// TIA Portal V19 export
FUNCTION "FC_Rez_to_DB45" : Void   // FC1, LAD
TITLE = Füllt nach Aufgabetaste (Panel) Technologie DB
{ S7_Optimized_Access := 'TRUE' }
// stored: SetENOAutomatically true
   VAR_TEMP
      Ptr_Befehl_dyn : Int;
      Ptr_Param_dyn : Int;
      i : Int;
   END_VAR
   VAR CONSTANT
      KS : USInt := 1;   // kurz schmal
      LS : USInt := 2;   // lang schmal
      GO : USInt := 3;   // Großoptik
      Typ_KS : Byte := 16#11;
      Typ_LS : Byte := 16#12;
      Typ_GO : Byte := 16#20;
      Startpos_CM01 : Byte := 16#1;
      Startpos_CM02 : Byte := 16#D;
      Startpos_CM03 : Byte := 16#7;
      Startpos_CM04 : Byte := 16#13;
      Startpos_BE : Byte := 16#19;
      Laenge : Byte := 16#6;
      leer : Byte;
      M_area : Byte := 16#83;
      DB_area : Byte := 16#84;
      Ptr_Befehl_1 : Int := 260;   // Adresse Befehlsparameter
      Ptr_Befehl_2 : Int := 264;   // Adresse Befehlsparameter
      Ptr_Befehl_3 : Int := 268;   // Adresse Befehlsparameter
      Ptr_Befehl_4 : Int := 272;   // Adresse Befehlsparameter
      Ptr_Befehl_5 : Int := 276;   // Adresse Befehlsparameter
      Ptr_Befehl_6 : Int := 280;   // Adresse Befehlsparameter
      Ptr_Befehl_7 : Int;   // Adresse Befehlsparameter
      Techno_DB : DInt := 45;
   END_VAR
BEGIN

REGION Network 1 (SCL): aktuelle Auswahl in Arbeitsstruktur kopieren
   IF "DB_Prog_edit".akt_Aufgabe_Prog <> "DB_Prog_edit".old_Aufgabe_Prog THEN
       "DB_Prog_edit".Prog_Aufgabe.Prog := "DB_Prog_edit".Prog["DB_Prog_edit".akt_Aufgabe_Prog];

       "DB_Prog_edit".old_Aufgabe_Prog := "DB_Prog_edit".akt_Aufgabe_Prog;
   END_IF;
END_REGION

REGION Network 2 (SCL): Artikeldaten für aufgabe aufbereiten
   IF "Panel".Aufgabe.Freigabe AND "DB_Prog_edit".StandNr <> 0  AND "DB_Prog_edit".akt_Aufgabe_Prog <>0  AND "DB_Prog_edit".Prog_Aufgabe.Korb_Nr <>0 THEN

       "DB_Prog_edit".GZ_Charge := "DB_Prog_edit".GZ_Charge + 1; // Gesamtzähler erhöhen
       "DB_Techno".WT_NR_lng := "DB_Prog_edit".GZ_Charge; // Chargenzähler
       "DB_Techno".STAND_NR := "DB_Prog_edit".StandNr; // Nummer B/E-Stand: 1..6
       "DB_Techno".Korb_Nr := INT_TO_USINT("DB_Prog_edit".Prog_Aufgabe.Korb_Nr); // Korb 1..13

       // Modus auswerten
       IF NOT "DB_ANLAGE".config.NormalB THEN
           // Kombi-Mode
           CASE "DB_Prog_edit".Prog_Aufgabe.Korb_Nr OF
               1..3:  // "151" Korb kurz 1..3
                   "DB_Prog_edit".Prog_Aufgabe.Prog.ParaByte.%X4 := TRUE;
                   "DB_Prog_edit".Prog_Aufgabe.Prog.ParaByte.%X5 := FALSE;

               4..8:   // "161" Korb kurz 4..8
                   "DB_Prog_edit".Prog_Aufgabe.Prog.ParaByte.%X4 := FALSE;
                   "DB_Prog_edit".Prog_Aufgabe.Prog.ParaByte.%X5 := TRUE;

               9..11:  // "151" Korb lang 1..3
                   "DB_Prog_edit".Prog_Aufgabe.Prog.ParaByte.%X4 := TRUE;
                   "DB_Prog_edit".Prog_Aufgabe.Prog.ParaByte.%X5 := FALSE;

               12..13:   // "161" Korb lang 4, Großoptik 
                   "DB_Prog_edit".Prog_Aufgabe.Prog.ParaByte.%X4 := FALSE;
                   "DB_Prog_edit".Prog_Aufgabe.Prog.ParaByte.%X5 := TRUE;
           END_CASE;

       ELSE
           // Normalbetrieb
           "DB_Prog_edit".Prog_Aufgabe.Prog.ParaByte.%X4 := FALSE;
           "DB_Prog_edit".Prog_Aufgabe.Prog.ParaByte.%X5 := FALSE;
       END_IF;

       "DB_Techno".Technologie := "DB_Prog_edit".akt_Aufgabe_Prog; // aktuelles Programm: 1..99
           // WT-Typ
       CASE "DB_Prog_edit".Prog_Aufgabe.Prog.Geometrie OF
           #KS:  
               "DB_Techno".WT_Typ := #Typ_KS;
           #LS:  
               "DB_Techno".WT_Typ := #Typ_LS;
           #GO:
               "DB_Techno".WT_Typ := #Typ_GO;
           ELSE
               "DB_Techno".WT_Typ := 0;
       END_CASE;
    // Langsam senken /Langsam heben / Modi
       "DB_Techno".ParaByte := "DB_Prog_edit".Prog_Aufgabe.Prog.ParaByte;

       "DB_Techno".KorrATZ := "DB_Prog_edit".Prog_Aufgabe.Prog.Faktor_ATZ;
       "DB_Techno".KorrPend := 1.0;


       // Normal-Betrieb - nur Ware "151" Gruppe CM01/CM02
       IF "DB_ANLAGE".config.NormalB THEN
           REGION NormalB
               // Vorspülen
               #Ptr_Befehl_dyn := 1;
               #Ptr_Param_dyn := 340;

               "DB_Techno".stBefehle[#Ptr_Befehl_dyn].Kennung := #Startpos_CM03;
               "DB_Techno".stBefehle[#Ptr_Befehl_dyn].FirstPos1 := #Startpos_CM03;
               "DB_Techno".stBefehle[#Ptr_Befehl_dyn].Grpleng1 := #Laenge;
               "DB_Techno".stBefehle[#Ptr_Befehl_dyn].FirstPos2 := #leer;
               "DB_Techno".stBefehle[#Ptr_Befehl_dyn].Grpleng2 := #leer;
               "DB_Techno".stBefehle[#Ptr_Befehl_dyn].Merker := #leer;
               "DB_Techno".stBefehle[#Ptr_Befehl_dyn].Param_Ptr := #Ptr_Param_dyn; //#Ptr_Befehl_1;
               "temp_Sollzeit" := TOD_TO_DINT("DB_Prog_edit".Prog_Aufgabe.Prog.CM03_VorSpuel.Expo) / 1000;

               POKE_BLK(area_src := #M_area,
                        dbNumber_src := 0,
                        byteOffset_src := 256,
                        area_dest := #DB_area,
                        dbNumber_dest := #Techno_DB,
                        byteOffset_dest := #Ptr_Param_dyn, //Ptr_Befehl_1,
                        count := 4);

               // Vorätzen
               IF "DB_Prog_edit".Prog_Aufgabe.Prog.CM01_VorAetz.Anzahl_Voraetz > 0 THEN
                   FOR #i := 1 TO BYTE_TO_INT("DB_Prog_edit".Prog_Aufgabe.Prog.CM01_VorAetz.Anzahl_Voraetz) DO
                       #Ptr_Befehl_dyn := #Ptr_Befehl_dyn + 1;
                       #Ptr_Param_dyn := #Ptr_Param_dyn + 4;

                       "DB_Techno".stBefehle[#Ptr_Befehl_dyn].Kennung := #Startpos_CM01;
                       "DB_Techno".stBefehle[#Ptr_Befehl_dyn].FirstPos1 := #Startpos_CM01;
                       "DB_Techno".stBefehle[#Ptr_Befehl_dyn].Grpleng1 := #Laenge;
                       "DB_Techno".stBefehle[#Ptr_Befehl_dyn].FirstPos2 := #Startpos_CM02;
                       "DB_Techno".stBefehle[#Ptr_Befehl_dyn].Grpleng2 := #Laenge;
                       "DB_Techno".stBefehle[#Ptr_Befehl_dyn].Merker := #leer;
                       "DB_Techno".stBefehle[#Ptr_Befehl_dyn].Param_Ptr := #Ptr_Param_dyn; // #Ptr_Befehl_2;
                       "temp_Sollzeit" := TOD_TO_DINT("DB_Prog_edit".Prog_Aufgabe.Prog.CM01_VorAetz.Expo) / 1000;

                       POKE_BLK(area_src := #M_area,
                                dbNumber_src := 0,
                                byteOffset_src := 256,
                                area_dest := #DB_area,
                                dbNumber_dest := #Techno_DB,
                                byteOffset_dest := #Ptr_Param_dyn, //Ptr_Befehl_2,
                                count := 4);


                       // Spülen Vorätzen
                       #Ptr_Befehl_dyn := #Ptr_Befehl_dyn + 1;
                       #Ptr_Param_dyn := #Ptr_Param_dyn + 4;

                       "DB_Techno".stBefehle[#Ptr_Befehl_dyn].Kennung := #Startpos_CM03;
                       "DB_Techno".stBefehle[#Ptr_Befehl_dyn].FirstPos1 := #Startpos_CM03;
                       "DB_Techno".stBefehle[#Ptr_Befehl_dyn].Grpleng1 := #Laenge;
                       "DB_Techno".stBefehle[#Ptr_Befehl_dyn].FirstPos2 := #leer;
                       "DB_Techno".stBefehle[#Ptr_Befehl_dyn].Grpleng2 := #leer;
                       "DB_Techno".stBefehle[#Ptr_Befehl_dyn].Merker := #leer;
                       "DB_Techno".stBefehle[#Ptr_Befehl_dyn].Param_Ptr := #Ptr_Param_dyn; // #Ptr_Befehl_3;
                       "temp_Sollzeit" := TOD_TO_DINT("DB_Prog_edit".Prog_Aufgabe.Prog.CM03_SpuelVorAetz.Expo) / 1000;

                       POKE_BLK(area_src := #M_area,
                                dbNumber_src := 0,
                                byteOffset_src := 256,
                                area_dest := #DB_area,
                                dbNumber_dest := #Techno_DB,
                                byteOffset_dest := #Ptr_Param_dyn, //#Ptr_Befehl_3,
                                count := 4);

                   END_FOR;
               END_IF;

               // Ätzen
               #Ptr_Befehl_dyn := #Ptr_Befehl_dyn + 1;
               #Ptr_Param_dyn := #Ptr_Param_dyn + 4;

               "DB_Techno".stBefehle[#Ptr_Befehl_dyn].Kennung := #Startpos_CM01;
               "DB_Techno".stBefehle[#Ptr_Befehl_dyn].FirstPos1 := #Startpos_CM01;
               "DB_Techno".stBefehle[#Ptr_Befehl_dyn].Grpleng1 := #Laenge;
               "DB_Techno".stBefehle[#Ptr_Befehl_dyn].FirstPos2 := #Startpos_CM02;
               "DB_Techno".stBefehle[#Ptr_Befehl_dyn].Grpleng2 := #Laenge;
               "DB_Techno".stBefehle[#Ptr_Befehl_dyn].Merker := #leer;
               "DB_Techno".stBefehle[#Ptr_Befehl_dyn].Param_Ptr := #Ptr_Param_dyn; //#Ptr_Befehl_4;
               "temp_Sollzeit" := TOD_TO_DINT("DB_Prog_edit".Prog_Aufgabe.Prog.CM01_Aetzen.Expo) / 1000;

               POKE_BLK(area_src := #M_area,
                        dbNumber_src := 0,
                        byteOffset_src := 256,
                        area_dest := #DB_area,
                        dbNumber_dest := #Techno_DB,
                        byteOffset_dest := #Ptr_Param_dyn, //#Ptr_Befehl_4,
                        count := 4);

               // Spülen 1 Ätzen
               #Ptr_Befehl_dyn := #Ptr_Befehl_dyn + 1;
               #Ptr_Param_dyn := #Ptr_Param_dyn + 4;

               "DB_Techno".stBefehle[#Ptr_Befehl_dyn].Kennung := #Startpos_CM03;
               "DB_Techno".stBefehle[#Ptr_Befehl_dyn].FirstPos1 := #Startpos_CM03;
               "DB_Techno".stBefehle[#Ptr_Befehl_dyn].Grpleng1 := #Laenge;
               "DB_Techno".stBefehle[#Ptr_Befehl_dyn].FirstPos2 := #leer;
               "DB_Techno".stBefehle[#Ptr_Befehl_dyn].Grpleng2 := #leer;
               "DB_Techno".stBefehle[#Ptr_Befehl_dyn].Merker := #leer;
               "DB_Techno".stBefehle[#Ptr_Befehl_dyn].Param_Ptr := #Ptr_Param_dyn; //#Ptr_Befehl_5;
               "temp_Sollzeit" := TOD_TO_DINT("DB_Prog_edit".Prog_Aufgabe.Prog.CM03_Spl_1.Expo) / 1000;

               POKE_BLK(area_src := #M_area,
                        dbNumber_src := 0,
                        byteOffset_src := 256,
                        area_dest := #DB_area,
                        dbNumber_dest := #Techno_DB,
                        byteOffset_dest := #Ptr_Param_dyn, //#Ptr_Befehl_5,
                        count := 4);

               // Spülen 2 Ätzen
               #Ptr_Befehl_dyn := #Ptr_Befehl_dyn + 1;
               #Ptr_Param_dyn := #Ptr_Param_dyn + 4;

               "DB_Techno".stBefehle[#Ptr_Befehl_dyn].Kennung := #Startpos_CM04;
               "DB_Techno".stBefehle[#Ptr_Befehl_dyn].FirstPos1 := #Startpos_CM04;
               "DB_Techno".stBefehle[#Ptr_Befehl_dyn].Grpleng1 := #Laenge;
               "DB_Techno".stBefehle[#Ptr_Befehl_dyn].FirstPos2 := #leer;
               "DB_Techno".stBefehle[#Ptr_Befehl_dyn].Grpleng2 := #leer;
               "DB_Techno".stBefehle[#Ptr_Befehl_dyn].Merker := #leer;
               "DB_Techno".stBefehle[#Ptr_Befehl_dyn].Param_Ptr := #Ptr_Param_dyn; //#Ptr_Befehl_6;
               "temp_Sollzeit" := TOD_TO_DINT("DB_Prog_edit".Prog_Aufgabe.Prog.CM04_Spl_2.Expo) / 1000;

               POKE_BLK(area_src := #M_area,
                        dbNumber_src := 0,
                        byteOffset_src := 256,
                        area_dest := #DB_area,
                        dbNumber_dest := #Techno_DB,
                        byteOffset_dest := #Ptr_Param_dyn, //#Ptr_Befehl_6,
                        count := 4);
           END_REGION

       ELSE // Kombi-Modus: "151" CM02 / CM04 ; "161" CM01 / CM03


           IF  "DB_Prog_edit".Prog_Aufgabe.Prog.ParaByte.%X4 THEN
            REGION WT_151                    
                // Vorspülen             
                  #Ptr_Befehl_dyn := 1;
                  #Ptr_Param_dyn := 340;

                  "DB_Techno".stBefehle[#Ptr_Befehl_dyn].Kennung := #Startpos_CM04;
                   "DB_Techno".stBefehle[#Ptr_Befehl_dyn].FirstPos1 := #Startpos_CM04;
                   "DB_Techno".stBefehle[#Ptr_Befehl_dyn].Grpleng1 := #Laenge;
                   "DB_Techno".stBefehle[#Ptr_Befehl_dyn].FirstPos2 := #leer;
                   "DB_Techno".stBefehle[#Ptr_Befehl_dyn].Grpleng2 := #leer;
                   "DB_Techno".stBefehle[#Ptr_Befehl_dyn].Merker := #leer;
                   "DB_Techno".stBefehle[#Ptr_Befehl_dyn].Param_Ptr := #Ptr_Param_dyn; //#Ptr_Befehl_1;
                   "temp_Sollzeit" := TOD_TO_DINT("DB_Prog_edit".Prog_Aufgabe.Prog.CM03_VorSpuel.Expo) / 1000;

                   POKE_BLK(area_src := #M_area,
                            dbNumber_src := 0,
                            byteOffset_src := 256,
                            area_dest := #DB_area,
                            dbNumber_dest := #Techno_DB,
                            byteOffset_dest := #Ptr_Param_dyn, //Ptr_Befehl_1,
                            count := 4);

                   // Vorätzen
                   IF "DB_Prog_edit".Prog_Aufgabe.Prog.CM01_VorAetz.Anzahl_Voraetz > 0 THEN
                       FOR #i := 1 TO BYTE_TO_INT("DB_Prog_edit".Prog_Aufgabe.Prog.CM01_VorAetz.Anzahl_Voraetz) DO
                           #Ptr_Befehl_dyn := #Ptr_Befehl_dyn + 1;
                           #Ptr_Param_dyn := #Ptr_Param_dyn + 4;

                           "DB_Techno".stBefehle[#Ptr_Befehl_dyn].Kennung := #Startpos_CM02;
                           "DB_Techno".stBefehle[#Ptr_Befehl_dyn].FirstPos1 := #Startpos_CM02;
                           "DB_Techno".stBefehle[#Ptr_Befehl_dyn].Grpleng1 := #Laenge;
                           "DB_Techno".stBefehle[#Ptr_Befehl_dyn].FirstPos2 := #leer;
                           "DB_Techno".stBefehle[#Ptr_Befehl_dyn].Grpleng2 := #leer;
                           "DB_Techno".stBefehle[#Ptr_Befehl_dyn].Merker := #leer;
                           "DB_Techno".stBefehle[#Ptr_Befehl_dyn].Param_Ptr := #Ptr_Param_dyn; // #Ptr_Befehl_2;
                           "temp_Sollzeit" := TOD_TO_DINT("DB_Prog_edit".Prog_Aufgabe.Prog.CM01_VorAetz.Expo) / 1000;

                           POKE_BLK(area_src := #M_area,
                                    dbNumber_src := 0,
                                    byteOffset_src := 256,
                                    area_dest := #DB_area,
                                    dbNumber_dest := #Techno_DB,
                                    byteOffset_dest := #Ptr_Param_dyn, //Ptr_Befehl_2,
                                    count := 4);

                           // Spülen Vorätzen
                           #Ptr_Befehl_dyn := #Ptr_Befehl_dyn + 1;
                           #Ptr_Param_dyn := #Ptr_Param_dyn + 4;

                           "DB_Techno".stBefehle[#Ptr_Befehl_dyn].Kennung := #Startpos_CM04;
                           "DB_Techno".stBefehle[#Ptr_Befehl_dyn].FirstPos1 := #Startpos_CM04;
                           "DB_Techno".stBefehle[#Ptr_Befehl_dyn].Grpleng1 := #Laenge;
                           "DB_Techno".stBefehle[#Ptr_Befehl_dyn].FirstPos2 := #leer;
                           "DB_Techno".stBefehle[#Ptr_Befehl_dyn].Grpleng2 := #leer;
                           "DB_Techno".stBefehle[#Ptr_Befehl_dyn].Merker := #leer;
                           "DB_Techno".stBefehle[#Ptr_Befehl_dyn].Param_Ptr := #Ptr_Param_dyn; // #Ptr_Befehl_3;
                           "temp_Sollzeit" := TOD_TO_DINT("DB_Prog_edit".Prog_Aufgabe.Prog.CM03_SpuelVorAetz.Expo) / 1000;

                           POKE_BLK(area_src := #M_area,
                                    dbNumber_src := 0,
                                    byteOffset_src := 256,
                                    area_dest := #DB_area,
                                    dbNumber_dest := #Techno_DB,
                                    byteOffset_dest := #Ptr_Param_dyn, //#Ptr_Befehl_3,
                                    count := 4);

                       END_FOR;
                   END_IF;

                   // Ätzen
                   #Ptr_Befehl_dyn := #Ptr_Befehl_dyn + 1;
                   #Ptr_Param_dyn := #Ptr_Param_dyn + 4;

                   "DB_Techno".stBefehle[#Ptr_Befehl_dyn].Kennung := #Startpos_CM02;
                   "DB_Techno".stBefehle[#Ptr_Befehl_dyn].FirstPos1 := #Startpos_CM02;
                   "DB_Techno".stBefehle[#Ptr_Befehl_dyn].Grpleng1 := #Laenge;
                   "DB_Techno".stBefehle[#Ptr_Befehl_dyn].FirstPos2 := #leer;
                   "DB_Techno".stBefehle[#Ptr_Befehl_dyn].Grpleng2 := #leer;
                   "DB_Techno".stBefehle[#Ptr_Befehl_dyn].Merker := #leer;
                   "DB_Techno".stBefehle[#Ptr_Befehl_dyn].Param_Ptr := #Ptr_Param_dyn; //#Ptr_Befehl_4;
                   "temp_Sollzeit" := TOD_TO_DINT("DB_Prog_edit".Prog_Aufgabe.Prog.CM01_Aetzen.Expo) / 1000;

                   POKE_BLK(area_src := #M_area,
                            dbNumber_src := 0,
                            byteOffset_src := 256,
                            area_dest := #DB_area,
                            dbNumber_dest := #Techno_DB,
                            byteOffset_dest := #Ptr_Param_dyn, //#Ptr_Befehl_4,
                            count := 4);

                   // Spülen 1 Ätzen
                   #Ptr_Befehl_dyn := #Ptr_Befehl_dyn + 1;
                   #Ptr_Param_dyn := #Ptr_Param_dyn + 4;

                   "DB_Techno".stBefehle[#Ptr_Befehl_dyn].Kennung := #Startpos_CM04;
                   "DB_Techno".stBefehle[#Ptr_Befehl_dyn].FirstPos1 := #Startpos_CM04;
                   "DB_Techno".stBefehle[#Ptr_Befehl_dyn].Grpleng1 := #Laenge;
                   "DB_Techno".stBefehle[#Ptr_Befehl_dyn].FirstPos2 := #leer;
                   "DB_Techno".stBefehle[#Ptr_Befehl_dyn].Grpleng2 := #leer;
                   "DB_Techno".stBefehle[#Ptr_Befehl_dyn].Merker := #leer;
                   "DB_Techno".stBefehle[#Ptr_Befehl_dyn].Param_Ptr := #Ptr_Param_dyn; //#Ptr_Befehl_5;
                   "temp_Sollzeit" := TOD_TO_DINT("DB_Prog_edit".Prog_Aufgabe.Prog.CM03_Spl_1.Expo) / 1000;

                   POKE_BLK(area_src := #M_area,
                            dbNumber_src := 0,
                            byteOffset_src := 256,
                            area_dest := #DB_area,
                            dbNumber_dest := #Techno_DB,
                            byteOffset_dest := #Ptr_Param_dyn, //#Ptr_Befehl_5,
                            count := 4);

                   // Spülen 2 Ätzen
                   #Ptr_Befehl_dyn := #Ptr_Befehl_dyn + 1;
                   #Ptr_Param_dyn := #Ptr_Param_dyn + 4;

                   "DB_Techno".stBefehle[#Ptr_Befehl_dyn].Kennung := #Startpos_CM04;
                   "DB_Techno".stBefehle[#Ptr_Befehl_dyn].FirstPos1 := #Startpos_CM04;
                   "DB_Techno".stBefehle[#Ptr_Befehl_dyn].Grpleng1 := #Laenge;
                   "DB_Techno".stBefehle[#Ptr_Befehl_dyn].FirstPos2 := #leer;
                   "DB_Techno".stBefehle[#Ptr_Befehl_dyn].Grpleng2 := #leer;
                   "DB_Techno".stBefehle[#Ptr_Befehl_dyn].Merker := #leer;
                   "DB_Techno".stBefehle[#Ptr_Befehl_dyn].Param_Ptr := #Ptr_Param_dyn; //#Ptr_Befehl_6;
                   "temp_Sollzeit" := TOD_TO_DINT("DB_Prog_edit".Prog_Aufgabe.Prog.CM04_Spl_2.Expo) / 1000;

                   POKE_BLK(area_src := #M_area,
                            dbNumber_src := 0,
                            byteOffset_src := 256,
                            area_dest := #DB_area,
                            dbNumber_dest := #Techno_DB,
                            byteOffset_dest := #Ptr_Param_dyn, //#Ptr_Befehl_6,
                            count := 4);
               END_REGION

           ELSE
            REGION WT_161                    
                   // Vorspülen             
                   #Ptr_Befehl_dyn := 1;
                   #Ptr_Param_dyn := 340;

                   "DB_Techno".stBefehle[#Ptr_Befehl_dyn].Kennung := #Startpos_CM03;
                   "DB_Techno".stBefehle[#Ptr_Befehl_dyn].FirstPos1 := #Startpos_CM03;
                   "DB_Techno".stBefehle[#Ptr_Befehl_dyn].Grpleng1 := #Laenge;
                   "DB_Techno".stBefehle[#Ptr_Befehl_dyn].FirstPos2 := #leer;
                   "DB_Techno".stBefehle[#Ptr_Befehl_dyn].Grpleng2 := #leer;
                   "DB_Techno".stBefehle[#Ptr_Befehl_dyn].Merker := #leer;
                   "DB_Techno".stBefehle[#Ptr_Befehl_dyn].Param_Ptr := #Ptr_Param_dyn; //#Ptr_Befehl_1;
                   "temp_Sollzeit" := TOD_TO_DINT("DB_Prog_edit".Prog_Aufgabe.Prog.CM03_VorSpuel.Expo) / 1000;

                   POKE_BLK(area_src := #M_area,
                            dbNumber_src := 0,
                            byteOffset_src := 256,
                            area_dest := #DB_area,
                            dbNumber_dest := #Techno_DB,
                            byteOffset_dest := #Ptr_Param_dyn, //Ptr_Befehl_1,
                            count := 4);

                   // Vorätzen
                   IF "DB_Prog_edit".Prog_Aufgabe.Prog.CM01_VorAetz.Anzahl_Voraetz > 0 THEN
                       FOR #i := 1 TO BYTE_TO_INT("DB_Prog_edit".Prog_Aufgabe.Prog.CM01_VorAetz.Anzahl_Voraetz) DO
                           #Ptr_Befehl_dyn := #Ptr_Befehl_dyn + 1;
                           #Ptr_Param_dyn := #Ptr_Param_dyn + 4;

                           "DB_Techno".stBefehle[#Ptr_Befehl_dyn].Kennung := #Startpos_CM01;
                           "DB_Techno".stBefehle[#Ptr_Befehl_dyn].FirstPos1 := #Startpos_CM01;
                           "DB_Techno".stBefehle[#Ptr_Befehl_dyn].Grpleng1 := #Laenge;
                           "DB_Techno".stBefehle[#Ptr_Befehl_dyn].FirstPos2 := #leer;
                           "DB_Techno".stBefehle[#Ptr_Befehl_dyn].Grpleng2 := #leer;
                           "DB_Techno".stBefehle[#Ptr_Befehl_dyn].Merker := #leer;
                           "DB_Techno".stBefehle[#Ptr_Befehl_dyn].Param_Ptr := #Ptr_Param_dyn; // #Ptr_Befehl_2;
                           "temp_Sollzeit" := TOD_TO_DINT("DB_Prog_edit".Prog_Aufgabe.Prog.CM01_VorAetz.Expo) / 1000;

                           POKE_BLK(area_src := #M_area,
                                    dbNumber_src := 0,
                                    byteOffset_src := 256,
                                    area_dest := #DB_area,
                                    dbNumber_dest := #Techno_DB,
                                    byteOffset_dest := #Ptr_Param_dyn, //Ptr_Befehl_2,
                                    count := 4);

                           // Spülen Vorätzen
                           #Ptr_Befehl_dyn := #Ptr_Befehl_dyn + 1;
                           #Ptr_Param_dyn := #Ptr_Param_dyn + 4;

                           "DB_Techno".stBefehle[#Ptr_Befehl_dyn].Kennung := #Startpos_CM03;
                           "DB_Techno".stBefehle[#Ptr_Befehl_dyn].FirstPos1 := #Startpos_CM03;
                           "DB_Techno".stBefehle[#Ptr_Befehl_dyn].Grpleng1 := #Laenge;
                           "DB_Techno".stBefehle[#Ptr_Befehl_dyn].FirstPos2 := #leer;
                           "DB_Techno".stBefehle[#Ptr_Befehl_dyn].Grpleng2 := #leer;
                           "DB_Techno".stBefehle[#Ptr_Befehl_dyn].Merker := #leer;
                           "DB_Techno".stBefehle[#Ptr_Befehl_dyn].Param_Ptr := #Ptr_Param_dyn; // #Ptr_Befehl_3;
                           "temp_Sollzeit" := TOD_TO_DINT("DB_Prog_edit".Prog_Aufgabe.Prog.CM03_SpuelVorAetz.Expo) / 1000;

                           POKE_BLK(area_src := #M_area,
                                    dbNumber_src := 0,
                                    byteOffset_src := 256,
                                    area_dest := #DB_area,
                                    dbNumber_dest := #Techno_DB,
                                    byteOffset_dest := #Ptr_Param_dyn, //#Ptr_Befehl_3,
                                    count := 4);

                       END_FOR;
                   END_IF;

                   // Ätzen
                   #Ptr_Befehl_dyn := #Ptr_Befehl_dyn + 1;
                   #Ptr_Param_dyn := #Ptr_Param_dyn + 4;

                   "DB_Techno".stBefehle[#Ptr_Befehl_dyn].Kennung := #Startpos_CM01;
                   "DB_Techno".stBefehle[#Ptr_Befehl_dyn].FirstPos1 := #Startpos_CM01;
                   "DB_Techno".stBefehle[#Ptr_Befehl_dyn].Grpleng1 := #Laenge;
                   "DB_Techno".stBefehle[#Ptr_Befehl_dyn].FirstPos2 := #leer;
                   "DB_Techno".stBefehle[#Ptr_Befehl_dyn].Grpleng2 := #leer;
                   "DB_Techno".stBefehle[#Ptr_Befehl_dyn].Merker := #leer;
                   "DB_Techno".stBefehle[#Ptr_Befehl_dyn].Param_Ptr := #Ptr_Param_dyn; //#Ptr_Befehl_4;
                   "temp_Sollzeit" := TOD_TO_DINT("DB_Prog_edit".Prog_Aufgabe.Prog.CM01_Aetzen.Expo) / 1000;

                   POKE_BLK(area_src := #M_area,
                            dbNumber_src := 0,
                            byteOffset_src := 256,
                            area_dest := #DB_area,
                            dbNumber_dest := #Techno_DB,
                            byteOffset_dest := #Ptr_Param_dyn, //#Ptr_Befehl_4,
                            count := 4);

                   // Spülen 1 Ätzen
                   #Ptr_Befehl_dyn := #Ptr_Befehl_dyn + 1;
                   #Ptr_Param_dyn := #Ptr_Param_dyn + 4;

                   "DB_Techno".stBefehle[#Ptr_Befehl_dyn].Kennung := #Startpos_CM03;
                   "DB_Techno".stBefehle[#Ptr_Befehl_dyn].FirstPos1 := #Startpos_CM03;
                   "DB_Techno".stBefehle[#Ptr_Befehl_dyn].Grpleng1 := #Laenge;
                   "DB_Techno".stBefehle[#Ptr_Befehl_dyn].FirstPos2 := #leer;
                   "DB_Techno".stBefehle[#Ptr_Befehl_dyn].Grpleng2 := #leer;
                   "DB_Techno".stBefehle[#Ptr_Befehl_dyn].Merker := #leer;
                   "DB_Techno".stBefehle[#Ptr_Befehl_dyn].Param_Ptr := #Ptr_Param_dyn; //#Ptr_Befehl_5;
                   "temp_Sollzeit" := TOD_TO_DINT("DB_Prog_edit".Prog_Aufgabe.Prog.CM03_Spl_1.Expo) / 1000;

                   POKE_BLK(area_src := #M_area,
                            dbNumber_src := 0,
                            byteOffset_src := 256,
                            area_dest := #DB_area,
                            dbNumber_dest := #Techno_DB,
                            byteOffset_dest := #Ptr_Param_dyn, //#Ptr_Befehl_5,
                            count := 4);

                   // Spülen 2 Ätzen
                   #Ptr_Befehl_dyn := #Ptr_Befehl_dyn + 1;
                   #Ptr_Param_dyn := #Ptr_Param_dyn + 4;

                   "DB_Techno".stBefehle[#Ptr_Befehl_dyn].Kennung := #Startpos_CM03;
                   "DB_Techno".stBefehle[#Ptr_Befehl_dyn].FirstPos1 := #Startpos_CM03;
                   "DB_Techno".stBefehle[#Ptr_Befehl_dyn].Grpleng1 := #Laenge;
                   "DB_Techno".stBefehle[#Ptr_Befehl_dyn].FirstPos2 := #leer;
                   "DB_Techno".stBefehle[#Ptr_Befehl_dyn].Grpleng2 := #leer;
                   "DB_Techno".stBefehle[#Ptr_Befehl_dyn].Merker := #leer;
                   "DB_Techno".stBefehle[#Ptr_Befehl_dyn].Param_Ptr := #Ptr_Param_dyn; //#Ptr_Befehl_6;
                   "temp_Sollzeit" := TOD_TO_DINT("DB_Prog_edit".Prog_Aufgabe.Prog.CM04_Spl_2.Expo) / 1000;

                   POKE_BLK(area_src := #M_area,
                            dbNumber_src := 0,
                            byteOffset_src := 256,
                            area_dest := #DB_area,
                            dbNumber_dest := #Techno_DB,
                            byteOffset_dest := #Ptr_Param_dyn, //#Ptr_Befehl_6,
                            count := 4);
               END_REGION

            END_IF;

       END_IF;

       // Ausfahrt
       #Ptr_Befehl_dyn := #Ptr_Befehl_dyn + 1;
       #Ptr_Param_dyn := #Ptr_Param_dyn + 4;

       "DB_Techno".stBefehle[#Ptr_Befehl_dyn].Kennung := #Startpos_BE;
       "DB_Techno".stBefehle[#Ptr_Befehl_dyn].FirstPos1 := #Startpos_BE;
       "DB_Techno".stBefehle[#Ptr_Befehl_dyn].Grpleng1 := #Laenge;
       "DB_Techno".stBefehle[#Ptr_Befehl_dyn].FirstPos2 := #leer;
       "DB_Techno".stBefehle[#Ptr_Befehl_dyn].Grpleng2 := #leer;
       "DB_Techno".stBefehle[#Ptr_Befehl_dyn].Merker := #leer;
       "DB_Techno".stBefehle[#Ptr_Befehl_dyn].Param_Ptr := #Ptr_Param_dyn; //#Ptr_Befehl_7;

       // Ende
       #Ptr_Befehl_dyn := #Ptr_Befehl_dyn + 1;

       FOR #i := #Ptr_Befehl_dyn TO 20 DO
            #Ptr_Befehl_dyn := #i;
            // #Ptr_Param_dyn := #Ptr_Param_dyn + 4;

           "DB_Techno".stBefehle[#Ptr_Befehl_dyn].Kennung := #leer;
           "DB_Techno".stBefehle[#Ptr_Befehl_dyn].FirstPos1 := #leer;
           "DB_Techno".stBefehle[#Ptr_Befehl_dyn].Grpleng1 := #leer;
           "DB_Techno".stBefehle[#Ptr_Befehl_dyn].FirstPos2 := #leer;
           "DB_Techno".stBefehle[#Ptr_Befehl_dyn].Grpleng2 := #leer;
           "DB_Techno".stBefehle[#Ptr_Befehl_dyn].Merker := #leer;
           "DB_Techno".stBefehle[#Ptr_Befehl_dyn].Param_Ptr := 0;
       END_FOR;

       "DB_Techno".Name := "DB_Prog_edit".Prog_Aufgabe.Prog.Name;

       "DB_Techno".DATEN_gueltig := "Panel".Aufgabe.Freigabe;
       // Rücksetzen
       "Panel".Aufgabe.Freigabe := FALSE;
       "DB_Prog_edit".StandNr := 0;
       "DB_Prog_edit".Variante := 0;
       "DB_Prog_edit".Prog_Aufgabe.Korb_Nr := 0;

   END_IF;
END_REGION
END_FUNCTION
